(* IEC 61131-3 sources: std_i2980_v2.06_cp053/Source/IMM/ieccontrol/InjectionGeneral (part 15) *)

(* ---- ABMovePVCalib.pu ---- *)
(*
@h    ! WARNING !
@h    The Kemro K2 system (including software) only meets category B according to EN 954-1,
@h    thus it is not intended for usage in safety-relevant control applications in the field
@h    of personal safety (e.g. emergency stop).
@h    To implement potentially necessary safety-relevant control tasks, always use additional
@h    external safety devices that are intended for the particular purpose, and meet the necessary
@h    functional safety.
@h    For further information see EN 954-1 (EN ISO 13849-1) and/or the K2-x00 user manual, chapter
@h    "CE conformity, directives and standards".

In this AB the inject movements are realized.
This means inject movement with cutoff detection, inject movement in setup mode,
calibration for screw transducer (forward) and also the inject movement for auto purging

@FunctionID: S_KPIEC_PRINJ_01
@FunctionID: S_KPIEC_PRINJ_02
@FunctionID: S_KPIEC_CALTRANS_04

*)

IMPORT_OVER_LISTFILE
 GET_MY_FU_NAME
, SET_ALARM
, FCalculateCylinderSize
, FCalcScrewSize
, cLockGroupHeatingNozzle
, cLockGroupSafetyGateNozzle
, cLockGroupSafetyGateMold
, cLockGroupMotor
, nActive
, nInactive
, nSetup
, tnCalibState_Aborted
, tnCalibState_Error
, cValueChangeDuringCalibTooLow
, cMovePVCalib
, MAX_VOLTAGE
, cMoveBwd
, tnOperationMode
, tsVelPre
, tsMoveData
, KAPPL_LintabData3D
, KCTRL_Stable_Param
, tsCylinderData
, tsTraceLevel
, tsMoveCtrl
, ABPumpPressureVelocityCalib
, tsPumpCalibError
, tyCalibDevices
, tsDeviceId
, tyPumpData
, ABMovementRegister
, FBSetMovementState

END_IMPORT

ALGORITHM_BLOCK ABMovePVCalib #DUMMY_EDIT_BLOCK

SYSTEM_VAR
 sv_OperationMode : tnOperationMode;
 sv_rPressure : REAL;
 sv_rVelocity : REAL;
 sv_bOutputActive : BOOL (* Output is active *);
 sv_bPreOutputReady : BOOL (* PreOutput is ready *);
 sv_bTransducerError : BOOL;
 sv_bDoPumpPressureCalib : BOOL;
 sv_bDoPumpVelocityCalib : BOOL;
 sv_ConstPumpPressureVelocCalib : tsVelPre;
 sv_rScrewVelocity : REAL;
 sv_MovePVCalib : tsMoveData;
 sv_rActPressureHydr : REAL;
 sv_TmpLintab : KAPPL_LintabData3D;
 sv_rServoOutput : REAL;
 sv_ConstServoPressureVelocCalib : tsVelPre;
 sv_bPumpPreVelCalibAnotherStepN : BOOL;
 sv_bPumpPreVelCalibDone : BOOL;
 sv_rScrewPosition : REAL;
 sv_PressureStableParam : KCTRL_Stable_Param;
 sv_VelocityStableParam : KCTRL_Stable_Param;
 sv_CylinderData : tsCylinderData;
 sv_rScrewDiameter : REAL;
 sv_rTmpMaxAbsFlow : REAL;
 sv_TraceLevel : tsTraceLevel;
 sv_rScrewVolume : REAL;
 sv_rMaxVoltageVelocityPresCalib : REAL;
 sv_rMaxMeasurePositionRel : REAL;
 sv_PumpCalibError : tsPumpCalibError;
 sv_PumpCalibDevices : tyCalibDevices (* !!! device 1 - 20 reserved !!! *);
 sv_MoveDecompAftPlast : tsMoveData;
 sv_MoveInject : tsMoveData;
 sv_rScrewVelocityAbs : REAL (* screw velocity in mm/s *);
 sv_DeviceId : tsDeviceId;
 ai_Pressure : REAL;
 ai_SysPressure : REAL;
 sv_iCalibratingPump : DINT (* number of pump which is actually calibrating *);
 sv_PumpData : tyPumpData;
END_VAR

SYSTEM_OBJECT
 TaskInject : TASK;
 erSetupModeRequiredForCalib : ALARM;
END_OBJECT

VAR_EXTERNAL
 g_MoveCtrl : tsMoveCtrl;
END_VAR

VAR
 abPumpPressureVelocityCalib : ABPumpPressureVelocityCalib;
END_VAR

(*
This algorithm is necessary for registering the available movements
and the according parameters (Lockgroups, icon path, delay time, ....)
*)

ALGORITHM aRegister

VAR
 abInjectRegister : ABMovementRegister;
END_VAR
#BEGIN_EDIT_BLOCK
(**************************************** WARNING ********************************************
 *** The KEBA Kemro K2 System including software is not intended for safety control tasks! ***
 ***                       For further information see Comment tab!                        ***
 *********************************************************************************************)

//register inject movement
sv_MovePVCalib.LockGroups[1] := cLockGroupHeatingNozzle;
sv_MovePVCalib.LockGroups[2] := cLockGroupSafetyGateNozzle;
sv_MovePVCalib.LockGroups[3] := cLockGroupSafetyGateMold;
sv_MovePVCalib.LockGroups[4] := cLockGroupMotor;
sv_MovePVCalib.sIconPath := CONCAT(GET_MY_FU_NAME(),"\hmi\images\movScrewFwd.gif");

abInjectRegister.aRegister(@sv_MovePVCalib);

;#END_EDIT_BLOCK END_ALGORITHM

(*
This algorithm is responsible for executing the movement.
Depending on MoveId, OperationMode and activated transducer calibration the according
movement is executed.
The different actions contain the movement blocks and the according parameters.
*)

ALGORITHM aRun

VAR_INPUT
 bStop : BOOL (* flag if the movement should be stopped *);
END_VAR

VAR_OUTPUT
 bReady : BOOL (* information if movement is ready *);
END_VAR

VAR
 fbSetMovementState : FBSetMovementState;
 bError : BOOL;
 rSizeHydraulicCylinder : REAL;
 rSizeScrewCylinder : REAL;
 rTmpMaxAbsVel : REAL;
 iLastCalibratedPump : DINT;
END_VAR

(* IecGraph-Code *)

(* init step *)
INITIAL_STEP START:
AStart (P);
END_STEP

ACTION AStart: #BEGIN_EDIT_BLOCK
bReady := FALSE;
fbSetMovementState(MoveId   := g_MoveCtrl.pData^.MoveId,
                   MoveDir  := g_MoveCtrl.pData^.MoveDir,
                   State    := nActive);

;#END_EDIT_BLOCK END_ACTION (*AStart*)

(* steps *)
STEP S_InitMaxVoltage:
AInit (P);
END_STEP

STEP S_NotInSetupMode:
ANotInSetupMode (P);
END_STEP

ACTION ANotInSetupMode: #BEGIN_EDIT_BLOCK
SET_ALARM(erSetupModeRequiredForCalib);

;#END_EDIT_BLOCK END_ACTION (*ANotInSetupMode*)
STEP S_InjectPresVelCalib:
AResetCalibPressureVelocity (P);
APressureVelocityCalib (N);
ACalc (P0);
END_STEP

STEP S_Ready:
AReady (P);
END_STEP

ACTION AReady: #BEGIN_EDIT_BLOCK
bReady := TRUE;
fbSetMovementState(MoveId   := g_MoveCtrl.pData^.MoveId,
                   MoveDir  := g_MoveCtrl.pData^.MoveDir,
                   State    := nInactive);

;#END_EDIT_BLOCK END_ACTION (*AReady*)

(* transitions *)
GO_ON_TRANSITION TSetupMode (* TSetupMode *) FROM START TO S_InitMaxVoltage :=  #BEGIN_EDIT_BLOCK
sv_OperationMode = nSetup

;#END_EDIT_BLOCK
END_TRANSITION

TRANSITION Trans6 (* Trans6 *) FROM S_InitMaxVoltage TO S_InjectPresVelCalib :=  #BEGIN_EDIT_BLOCK
TRUE
;#END_EDIT_BLOCK
END_TRANSITION

GO_ON_TRANSITION TNotSetupMode (* TNotSetupMode *) FROM START TO S_NotInSetupMode :=  #BEGIN_EDIT_BLOCK
sv_OperationMode <> nSetup
;#END_EDIT_BLOCK
END_TRANSITION

GO_ON_TRANSITION Trans35 (* Trans35 *) FROM S_NotInSetupMode TO S_Ready :=  #BEGIN_EDIT_BLOCK
TRUE
;#END_EDIT_BLOCK
END_TRANSITION

TRANSITION TPVCalibDone (* TPVCalibDone *) FROM S_InjectPresVelCalib TO S_Ready :=  #BEGIN_EDIT_BLOCK
NOT abPumpPressureVelocityCalib.aRun.bActive
;#END_EDIT_BLOCK
END_TRANSITION

TRANSITION TReady (* TReady *) FROM S_Ready TO START :=  #BEGIN_EDIT_BLOCK
TRUE
;#END_EDIT_BLOCK
END_TRANSITION

(* end IecGraph-Code *)
(* sfc-code *)

(* stand alone actions *)
ACTION AResetCalibPressureVelocity: #BEGIN_EDIT_BLOCK
(**************************************** WARNING ********************************************
 *** The KEBA Kemro K2 System including software is not intended for safety control tasks! ***
 ***                       For further information see Comment tab!                        ***
 *********************************************************************************************)

bError := FALSE;
abPumpPressureVelocityCalib.aRun(bStart := FALSE);

;#END_EDIT_BLOCK END_ACTION (*AResetCalibPressureVelocity*)
ACTION ACalc: #BEGIN_EDIT_BLOCK
(**************************************** WARNING ********************************************
 *** The KEBA Kemro K2 System including software is not intended for safety control tasks! ***
 ***                       For further information see Comment tab!                        ***
 *********************************************************************************************)

IF sv_bPumpPreVelCalibDone AND NOT bError THEN
   rSizeHydraulicCylinder := FCalculateCylinderSize(CylinderData := sv_CylinderData, bSmallSize := sv_CylinderData.bUseSmallSize, bCalcHighPressSize := FALSE);
   rSizeScrewCylinder := FCalcScrewSize(rDiameter := sv_rScrewDiameter);

   // convert velocity from [cm^3/s] to [mm/s]
   rTmpMaxAbsVel := abPumpPressureVelocityCalib.aRun.rMaxVelocityAbs * 1000.0 / rSizeScrewCylinder;

   // convert velocity from [mm/s] to [l/min] in hydraulic volume
   sv_rTmpMaxAbsFlow := rTmpMaxAbsVel * rSizeHydraulicCylinder / 1000000.0 * 60.0;
END_IF;

;#END_EDIT_BLOCK END_ACTION (*ACalc*)
ACTION APressureVelocityCalib: #BEGIN_EDIT_BLOCK
(**************************************** WARNING ********************************************
 *** The KEBA Kemro K2 System including software is not intended for safety control tasks! ***
 ***                       For further information see Comment tab!                        ***
 *********************************************************************************************)

//output pressure in bar, velocity in % of Pump
abPumpPressureVelocityCalib.aRun(bStop := bStop OR sv_bTransducerError,
                                 bStart := TRUE,
                                 rActPosition := sv_rScrewPosition,
                                 rMaxPosition := sv_rScrewVolume,
                                 rActVel := sv_rScrewVelocity,
                                 rActPressure := sv_rActPressureHydr,
                                 bIsPressureCalib := sv_bDoPumpPressureCalib,
                                 bIsVelocityCalib := sv_bDoPumpVelocityCalib,
                                 bIsServoValveCalib := FALSE,
                                 bDirection := FALSE,
                                 dDelayTimePump := T#200ms,
                                 rLimitPositionFactor := sv_rMaxMeasurePositionRel,
                                 bActive => sv_bOutputActive,
                                 rOutputPre => sv_rPressure,
                                 rOutputVel => sv_rVelocity,
                                 rOutputServo => sv_rServoOutput,
                                 bPreOutputReached => sv_bPreOutputReady,
                                 bError => sv_PumpCalibError.bError,
                                 iErrorInfo => sv_PumpCalibError.iErrorInfo);

;#END_EDIT_BLOCK END_ACTION (*APressureVelocityCalib*)
ACTION AInit: #BEGIN_EDIT_BLOCK
(**************************************** WARNING ********************************************
 *** The KEBA Kemro K2 System including software is not intended for safety control tasks! ***
 ***                       For further information see Comment tab!                        ***
 *********************************************************************************************)

IF iLastCalibratedPump <> sv_iCalibratingPump THEN
   //get max voltages of the pump which should be calibrated
   abPumpPressureVelocityCalib.aInitMaxVoltages.rMaxVoltage := MAX_VOLTAGE;
   abPumpPressureVelocityCalib.aInitMaxVoltages.rMinVoltage := 0.0;
   abPumpPressureVelocityCalib.aInitMaxVoltages.prMaxVoltageVelocity := sv_PumpData[sv_iCalibratingPump].prMaxVoltageV;
   abPumpPressureVelocityCalib.aInitMaxVoltages.prMaxVoltagePressure := sv_PumpData[sv_iCalibratingPump].prMaxVoltageP;
   abPumpPressureVelocityCalib.aInitMaxVoltages.prMaxVoltageVelocityPresCalib := @sv_rMaxVoltageVelocityPresCalib;
   abPumpPressureVelocityCalib.aInitMaxVoltages();

   iLastCalibratedPump := sv_iCalibratingPump;
END_IF;

;#END_EDIT_BLOCK END_ACTION (*AInit*)
(* end sfc-code *)

END_ALGORITHM

ALGORITHM aInit

VAR_TEMP
 i : DINT;
END_VAR
#BEGIN_EDIT_BLOCK
(**************************************** WARNING ********************************************
 *** The KEBA Kemro K2 System including software is not intended for safety control tasks! ***
 ***                       For further information see Comment tab!                        ***
 *********************************************************************************************)

abPumpPressureVelocityCalib.aInit(pConst := @sv_ConstPumpPressureVelocCalib,
                                  pConstServo := @sv_ConstServoPressureVelocCalib,
                                  MoveId := cMovePVCalib,
                                  pTmpLintab := @sv_TmpLintab,
                                  pbPumpPreVelCalibAnotherStepN := @sv_bPumpPreVelCalibAnotherStepN,
                                  pbPumpPreVelCalibDone := @sv_bPumpPreVelCalibDone,
                                  pPressureStableParam := @sv_PressureStableParam,
                                  pVelocityStableParam := @sv_VelocityStableParam,
                                  debugInstanceName := 'PVCalib',
                                  debugTask := TaskInject,
                                  pbDebugCalibration := @sv_TraceLevel.bDebugCalibration);

//add calib information to sv_PumpCalibDevices - list
FOR i := 1 TO cMaxCalibDevices DO
   IF sv_PumpCalibDevices[i].DeviceId = sv_DeviceId THEN
      sv_PumpCalibDevices[i].pVelCalibStartPosMovement := @sv_MoveDecompAftPlast;
      sv_PumpCalibDevices[i].pVelCalibMovement := @sv_MovePVCalib;
      sv_PumpCalibDevices[i].pPresCalibStartPosMovement := @sv_MoveInject;
      sv_PumpCalibDevices[i].pPresCalibMovement := @sv_MovePVCalib;
      sv_PumpCalibDevices[i].prActVelocity := @sv_rScrewVelocityAbs;
      IF IS_LINKED(ai_Pressure) OR IS_LINKED(ai_SysPressure) THEN
         sv_PumpCalibDevices[i].prActPressure := @sv_rActPressureHydr;
      END_IF;
      EXIT;
   END_IF;
END_FOR;

;#END_EDIT_BLOCK END_ALGORITHM

END_ALGORITHM_BLOCK

#END_OF_IEC_PART

@Puma @IecEditor 6 120 @Pou 25
@@@BEG_Comment@@@
@h    ! WARNING !
@h    The Kemro K2 system (including software) only meets category B according to EN 954-1,
@h    thus it is not intended for usage in safety-relevant control applications in the field
@h    of personal safety (e.g. emergency stop).
@h    To implement potentially necessary safety-relevant control tasks, always use additional
@h    external safety devices that are intended for the particular purpose, and meet the necessary
@h    functional safety.
@h    For further information see EN 954-1 (EN ISO 13849-1) and/or the K2-x00 user manual, chapter
@h    "CE conformity, directives and standards".

In this AB the inject movements are realized.
This means inject movement with cutoff detection, inject movement in setup mode,
calibration for screw transducer (forward) and also the inject movement for auto purging

@FunctionID: S_KPIEC_PRINJ_01
@FunctionID: S_KPIEC_PRINJ_02
@FunctionID: S_KPIEC_CALTRANS_04

@@@END_Comment@@@

@BEG_Contents

@BEG_Func
@RT(17)FuncTreeContainer
4
@Var @RT(14)GET_MY_FU_NAME @RT(0) @T @T @DERIVED 0 @F @RT(22)KEBA_STANDARD_FUNCTION @F
@T
@BEG_Attrib
0 @RT(0) @RT(0)
@END_Attrib
1 1 @F @F @F @F

@Var @RT(9)SET_ALARM @RT(0) @T @T @DERIVED 0 @F @RT(23)KEBA_STANDARD_PROCEDURE @F
@T
@BEG_Attrib
0 @RT(0) @RT(0)
@END_Attrib
1 1 @F @F @F @F

@Var @RT(22)FCalculateCylinderSize @RT(0) @T @T @DERIVED 0 @F @RT(8)FUNCTION @F
@T
@BEG_Attrib
0 @RT(0) @RT(0)
@END_Attrib
1 1 @F @F @F @F

@Var @RT(14)FCalcScrewSize @RT(0) @T @T @DERIVED 0 @F @RT(8)FUNCTION @F
@T
@BEG_Attrib
0 @RT(0) @RT(0)
@END_Attrib
1 1 @F @F @F @F

@END_Func

@BEG_Const
@RT(18)ConstTreeContainer
13
@Var @RT(23)cLockGroupHeatingNozzle @RT(0) @T @F @DT @RT(4)DINT @RT(0) @T @T @BASIC 0 @F
@F @F
@T
@BEG_Attrib
0 @RT(2)63 @RT(35)Members: Injection, Plast, Suckback
@END_Attrib
1 1 @F @F @F @F

@Var @RT(26)cLockGroupSafetyGateNozzle @RT(0) @T @F @DT @RT(4)DINT @RT(0) @T @T @BASIC 0 @F
@F @F
@T
@BEG_Attrib
0 @RT(2)62 @RT(59)Members: Nozzle Forward, Injection, Plast, Intrusion, Purge
@END_Attrib
1 1 @F @F @F @F

@Var @RT(24)cLockGroupSafetyGateMold @RT(0) @T @F @DT @RT(4)DINT @RT(0) @T @T @BASIC 0 @F
@F @F
@T
@BEG_Attrib
0 @RT(2)61 @RT(73)Members: Mold Close, Mold Hight Forward, Auto Mold Hight, Core In, Inject
@END_Attrib
1 1 @F @F @F @F

@Var @RT(15)cLockGroupMotor @RT(0) @T @F @DT @RT(4)DINT @RT(0) @T @T @BASIC 0 @F
@F @F
@T
@BEG_Attrib
0 @RT(2)69 @RT(56)Members: Mold, Ejector, Cores, Injection, Plast, Purge,
@END_Attrib
1 1 @F @F @F @F

@Var @RT(7)nActive @RT(0) @T @T @DERIVED 0 @F @RT(16)tnActiveInactive @F
@T
@BEG_Attrib
0 @RT(1)1 @RT(0)
@END_Attrib
1 1 @F @F @F @F

@Var @RT(9)nInactive @RT(0) @T @T @DERIVED 0 @F @RT(16)tnActiveInactive @F
@T
@BEG_Attrib
0 @RT(1)0 @RT(0)
@END_Attrib
1 1 @F @F @F @F

@Var @RT(6)nSetup @RT(0) @T @T @DERIVED 0 @F @RT(15)tnOperationMode @F
@T
@BEG_Attrib
0 @RT(1)0 @RT(36)Setup mode only for service engineer
@END_Attrib
1 1 @F @F @F @F

@Var @RT(20)tnCalibState_Aborted @RT(0) @T @T @DERIVED 0 @F @RT(12)tnCalibState @F
@T
@BEG_Attrib
0 @RT(1)4 @RT(19)calibration aborted
@END_Attrib
1 1 @F @F @F @F

@Var @RT(18)tnCalibState_Error @RT(0) @T @T @DERIVED 0 @F @RT(12)tnCalibState @F
@T
@BEG_Attrib
0 @RT(1)3 @RT(32)error occured during calibration
@END_Attrib
1 1 @F @F @F @F

@Var @RT(29)cValueChangeDuringCalibTooLow @RT(0) @T @F @DT @RT(4)DINT @RT(0) @T @T @BASIC 0 @F
@F @F
@T
@BEG_Attrib
0 @RT(4)-510 @RT(94)no or too low value change (velocity, pressure, rpm, ..) detected during calibration procedure
@END_Attrib
1 1 @F @F @F @F

@Var @RT(12)cMovePVCalib @RT(0) @T @F @DT @RT(4)DINT @RT(0) @T @T @BASIC 0 @F
@F @F
@T
@BEG_Attrib
0 @RT(2)38 @RT(38)injection movement with voltage output
@END_Attrib
1 1 @F @F @F @F

@Var @RT(11)MAX_VOLTAGE @RT(0) @T @F @DT @RT(4)REAL @RT(0) @T @T @BASIC 0 @F
@F @F
@T
@BEG_Attrib
0 @RT(4)10.0 @RT(0)
@END_Attrib
1 1 @F @F @F @F

@Var @RT(8)cMoveBwd @RT(0) @T @F @DT @RT(4)DINT @RT(0) @T @T @BASIC 0 @F
@F @F
@T
@BEG_Attrib
0 @RT(2)11 @RT(17)movement backward
@END_Attrib
1 1 @F @F @F @F

@END_Const

@BEG_Export

@BEG_Kind
@ALGORITHM_BLOCK @RT(13)ABMovePVCalib @STRUCTURED_TEXT
@RT(0) @RT(0) @RT(0)
@END_Kind

@BEG_Dcl
@RT(16)DclTreeContainer
41
@Var @RT(16)sv_OperationMode @RT(0) @T @T @DERIVED 0 @T @T @DT @RT(15)tnOperationMode @RT(0) @T @T @UNKNOWN 0 @F
@F @F
@T
@BEG_Attrib
3 @RT(0) @RT(0) @RT(0)
@END_Attrib
1 8 @F @F @F @F

@Var @RT(12)sv_rPressure @RT(0) @T @F @DT @RT(4)REAL @RT(0) @T @T @BASIC 0 @F
@F @F
@T
@BEG_Attrib
3 @RT(0) @RT(0) @RT(0)
@END_Attrib
1 8 @F @F @F @F

@Var @RT(12)sv_rVelocity @RT(0) @T @F @DT @RT(4)REAL @RT(0) @T @T @BASIC 0 @F
@F @F
@T
@BEG_Attrib
3 @RT(0) @RT(0) @RT(0)
@END_Attrib
1 8 @F @F @F @F

@Var @RT(16)sv_bOutputActive @RT(0) @T @F @DT @RT(4)BOOL @RT(0) @T @T @BASIC 0 @F
@F @F
@T
@BEG_Attrib
3 @RT(0) @RT(16)Output is active @RT(0)
@END_Attrib
1 8 @F @F @F @F

@Var @RT(18)sv_bPreOutputReady @RT(0) @T @F @DT @RT(4)BOOL @RT(0) @T @T @BASIC 0 @F
@F @F
@T
@BEG_Attrib
3 @RT(0) @RT(18)PreOutput is ready @RT(0)
@END_Attrib
1 8 @F @F @F @F

@Var @RT(19)sv_bTransducerError @RT(0) @T @F @DT @RT(4)BOOL @RT(0) @T @T @BASIC 0 @F
@F @F
@T
@BEG_Attrib
3 @RT(0) @RT(0) @RT(0)
@END_Attrib
1 8 @F @F @F @F

@Var @RT(23)sv_bDoPumpPressureCalib @RT(0) @T @F @DT @RT(4)BOOL @RT(0) @T @T @BASIC 0 @F
@F @F
@T
@BEG_Attrib
3 @RT(0) @RT(0) @RT(0)
@END_Attrib
1 8 @F @F @F @F

@Var @RT(23)sv_bDoPumpVelocityCalib @RT(0) @T @F @DT @RT(4)BOOL @RT(0) @T @T @BASIC 0 @F
@F @F
@T
@BEG_Attrib
3 @RT(0) @RT(0) @RT(0)
@END_Attrib
1 8 @F @F @F @F

@Var @RT(30)sv_ConstPumpPressureVelocCalib @RT(0) @T @T @DERIVED 0 @T @T @DT @RT(8)tsVelPre @RT(0) @T @T @UNKNOWN 0 @F
@F @F
@T
@BEG_Attrib
3 @RT(0) @RT(0) @RT(0)
@END_Attrib
1 8 @F @F @F @F

@Var @RT(17)sv_rScrewVelocity @RT(0) @T @F @DT @RT(4)REAL @RT(0) @T @T @BASIC 0 @F
@F @F
@T
@BEG_Attrib
3 @RT(0) @RT(0) @RT(0)
@END_Attrib
1 8 @F @F @F @F

@Var @RT(14)sv_MovePVCalib @RT(0) @T @T @DERIVED 0 @T @T @DT @RT(10)tsMoveData @RT(0) @T @T @UNKNOWN 0 @F
@F @F
@T
@BEG_Attrib
3 @RT(0) @RT(0) @RT(0)
@END_Attrib
1 8 @F @F @F @F

@Var @RT(19)sv_rActPressureHydr @RT(0) @T @F @DT @RT(4)REAL @RT(0) @T @T @BASIC 0 @F
@F @F
@T
@BEG_Attrib
3 @RT(0) @RT(0) @RT(0)
@END_Attrib
1 8 @F @F @F @F

@Var @RT(12)sv_TmpLintab @RT(0) @T @T @DERIVED 0 @T @T @DT @RT(18)KAPPL_LintabData3D @RT(0) @T @T @UNKNOWN 0 @F
@F @F
@T
@BEG_Attrib
3 @RT(0) @RT(0) @RT(0)
@END_Attrib
1 8 @F @F @F @F

@Var @RT(15)sv_rServoOutput @RT(0) @T @F @DT @RT(4)REAL @RT(0) @T @T @BASIC 0 @F
@F @F
@T
@BEG_Attrib
3 @RT(0) @RT(0) @RT(0)
@END_Attrib
1 8 @F @F @F @F

@Var @RT(31)sv_ConstServoPressureVelocCalib @RT(0) @T @T @DERIVED 0 @T @T @DT @RT(8)tsVelPre @RT(0) @T @T @UNKNOWN 0 @F
@F @F
@T
@BEG_Attrib
3 @RT(0) @RT(0) @RT(0)
@END_Attrib
1 8 @F @F @F @F

@Var @RT(31)sv_bPumpPreVelCalibAnotherStepN @RT(0) @T @F @DT @RT(4)BOOL @RT(0) @T @T @BASIC 0 @F
@F @F
@T
@BEG_Attrib
3 @RT(0) @RT(0) @RT(0)
@END_Attrib
1 8 @F @F @F @F

@Var @RT(23)sv_bPumpPreVelCalibDone @RT(0) @T @F @DT @RT(4)BOOL @RT(0) @T @T @BASIC 0 @F
@F @F
@T
@BEG_Attrib
3 @RT(0) @RT(0) @RT(0)
@END_Attrib
1 8 @F @F @F @F

@Var @RT(17)sv_rScrewPosition @RT(0) @T @F @DT @RT(4)REAL @RT(0) @T @T @BASIC 0 @F
@F @F
@T
@BEG_Attrib
3 @RT(0) @RT(0) @RT(0)
@END_Attrib
1 8 @F @F @F @F

@Var @RT(22)sv_PressureStableParam @RT(0) @T @T @DERIVED 0 @T @T @DT @RT(18)KCTRL_Stable_Param @RT(0) @T @T @UNKNOWN 0 @F
@F @F
@T
@BEG_Attrib
3 @RT(0) @RT(0) @RT(0)
@END_Attrib
1 8 @F @F @F @F

@Var @RT(22)sv_VelocityStableParam @RT(0) @T @T @DERIVED 0 @T @T @DT @RT(18)KCTRL_Stable_Param @RT(0) @T @T @UNKNOWN 0 @F
@F @F
@T
@BEG_Attrib
3 @RT(0) @RT(0) @RT(0)
@END_Attrib
1 8 @F @F @F @F

@Var @RT(15)sv_CylinderData @RT(0) @T @T @DERIVED 0 @T @T @DT @RT(14)tsCylinderData @RT(0) @T @T @UNKNOWN 0 @F
@F @F
@T
@BEG_Attrib
3 @RT(0) @RT(0) @RT(0)
@END_Attrib
1 8 @F @F @F @F

@Var @RT(17)sv_rScrewDiameter @RT(0) @T @F @DT @RT(4)REAL @RT(0) @T @T @BASIC 0 @F
@F @F
@T
@BEG_Attrib
3 @RT(0) @RT(0) @RT(0)
@END_Attrib
1 8 @F @F @F @F

@Var @RT(17)sv_rTmpMaxAbsFlow @RT(0) @T @F @DT @RT(4)REAL @RT(0) @T @T @BASIC 0 @F
@F @F
@T
@BEG_Attrib
3 @RT(0) @RT(0) @RT(0)
@END_Attrib
1 8 @F @F @F @F

@Var @RT(13)sv_TraceLevel @RT(0) @T @T @DERIVED 0 @T @T @DT @RT(12)tsTraceLevel @RT(0) @T @T @UNKNOWN 0 @F
@F @F
@T
@BEG_Attrib
3 @RT(0) @RT(0) @RT(0)
@END_Attrib
1 8 @F @F @F @F

@Var @RT(15)sv_rScrewVolume @RT(0) @T @F @DT @RT(4)REAL @RT(0) @T @T @BASIC 0 @F
@F @F
@T
@BEG_Attrib
3 @RT(0) @RT(0) @RT(0)
@END_Attrib
1 8 @F @F @F @F

@Var @RT(31)sv_rMaxVoltageVelocityPresCalib @RT(0) @T @F @DT @RT(4)REAL @RT(0) @T @T @BASIC 0 @F
@F @F
@T
@BEG_Attrib
3 @RT(0) @RT(0) @RT(0)
@END_Attrib
1 8 @F @F @F @F

@Var @RT(25)sv_rMaxMeasurePositionRel @RT(0) @T @F @DT @RT(4)REAL @RT(0) @T @T @BASIC 0 @F
@F @F
@T
@BEG_Attrib
3 @RT(0) @RT(0) @RT(0)
@END_Attrib
1 8 @F @F @F @F

@Var @RT(10)TaskInject @RT(0) @T @F @DT @RT(4)TASK @RT(0) @T @T @BASIC 0 @F
@F @F
@T
@BEG_Attrib
3 @RT(0) @RT(0) @RT(0)
@END_Attrib
1 7 @F @F @F @F

@Var @RT(27)erSetupModeRequiredForCalib @RT(0) @T @F @DT @RT(5)ALARM @RT(0) @T @T @BASIC 0 @F
@F @F
@T
@BEG_Attrib
3 @RT(0) @RT(0) @RT(0)
@END_Attrib
1 7 @F @F @F @F

@Var @RT(10)g_MoveCtrl @RT(0) @T @T @DERIVED 0 @T @T @DT @RT(10)tsMoveCtrl @RT(0) @T @T @UNKNOWN 0 @F
@F @F
@T
@BEG_Attrib
3 @RT(0) @RT(0) @RT(0)
@END_Attrib
1 6 @F @F @F @F

@Var @RT(27)abPumpPressureVelocityCalib @RT(0) @T @T @DERIVED 0 @T @T @DT @RT(27)ABPumpPressureVelocityCalib @RT(0) @T @T @UNKNOWN 0 @F
@F @F
@T
@BEG_Attrib
3 @RT(0) @RT(0) @RT(0)
@END_Attrib
1 0 @F @F @F @F

@Var @RT(17)sv_PumpCalibError @RT(0) @T @T @DERIVED 0 @T @T @DT @RT(16)tsPumpCalibError @RT(0) @T @T @UNKNOWN 0 @F
@F @F
@T
@BEG_Attrib
3 @RT(0) @RT(0) @RT(0)
@END_Attrib
1 8 @F @F @F @F

@Var @RT(19)sv_PumpCalibDevices @RT(0) @T @T @DERIVED 0 @T @T @DT @RT(14)tyCalibDevices @RT(0) @T @T @UNKNOWN 0 @F
@F @F
@T
@BEG_Attrib
3 @RT(0) @RT(30)!!! device 1 - 20 reserved !!! @RT(0)
@END_Attrib
1 8 @F @F @F @F

@Var @RT(21)sv_MoveDecompAftPlast @RT(0) @T @T @DERIVED 0 @T @T @DT @RT(10)tsMoveData @RT(0) @T @T @UNKNOWN 0 @F
@F @F
@T
@BEG_Attrib
3 @RT(0) @RT(0) @RT(0)
@END_Attrib
1 8 @F @F @F @F

@Var @RT(13)sv_MoveInject @RT(0) @T @T @DERIVED 0 @T @T @DT @RT(10)tsMoveData @RT(0) @T @T @UNKNOWN 0 @F
@F @F
@T
@BEG_Attrib
3 @RT(0) @RT(0) @RT(0)
@END_Attrib
1 8 @F @F @F @F

@Var @RT(20)sv_rScrewVelocityAbs @RT(0) @T @F @DT @RT(4)REAL @RT(0) @T @T @BASIC 0 @F
@F @F
@T
@BEG_Attrib
3 @RT(0) @RT(22)screw velocity in mm/s @RT(0)
@END_Attrib
1 8 @F @F @F @F

@Var @RT(11)sv_DeviceId @RT(0) @T @T @DERIVED 0 @T @T @DT @RT(10)tsDeviceId @RT(0) @T @T @UNKNOWN 0 @F
@F @F
@T
@BEG_Attrib
3 @RT(0) @RT(0) @RT(0)
@END_Attrib
1 8 @F @F @F @F

@Var @RT(11)ai_Pressure @RT(0) @T @F @DT @RT(4)REAL @RT(0) @T @T @BASIC 0 @F
@F @F
@T
@BEG_Attrib
3 @RT(0) @RT(0) @RT(0)
@END_Attrib
1 8 @F @F @F @F

@Var @RT(14)ai_SysPressure @RT(0) @T @F @DT @RT(4)REAL @RT(0) @T @T @BASIC 0 @F
@F @F
@T
@BEG_Attrib
3 @RT(0) @RT(0) @RT(0)
@END_Attrib
1 8 @F @F @F @F

@Var @RT(19)sv_iCalibratingPump @RT(0) @T @F @DT @RT(4)DINT @RT(0) @T @T @BASIC 0 @F
@F @F
@T
@BEG_Attrib
3 @RT(0) @RT(44)number of pump which is actually calibrating @RT(0)
@END_Attrib
1 8 @F @F @F @F

@Var @RT(11)sv_PumpData @RT(0) @T @T @DERIVED 0 @F @RT(10)tyPumpData @F
@T
@BEG_Attrib
3 @RT(0) @RT(0) @RT(0)
@END_Attrib
1 8 @F @F @F @F

@END_Dcl

@END_Export

@BEG_Body

3

@BEG_Export

@BEG_Algo
@ALGORITHM @RT(9)aRegister @STRUCTURED_TEXT
@RT(0) @RT(0) @RT(0) @F @F
@END_Algo

@BEG_Dcl
@RT(16)DclTreeContainer
1
@Var @RT(16)abInjectRegister @RT(0) @T @T @DERIVED 0 @T @T @DT @RT(18)ABMovementRegister @RT(0) @T @T @UNKNOWN 0 @F
@F @F
@T
@BEG_Attrib
3 @RT(0) @RT(0) @RT(0)
@END_Attrib
1 0 @F @F @F @F

@END_Dcl

@END_Export

@BEG_Export

@BEG_Algo
@ALGORITHM @RT(4)aRun @SEQUENTIAL_FLOW_CHART
@RT(0) @RT(0) @RT(0) @F @F
@END_Algo

@BEG_Dcl
@RT(16)DclTreeContainer
8
@Var @RT(5)bStop @RT(0) @T @F @DT @RT(4)BOOL @RT(0) @T @T @BASIC 0 @F
@F @F
@T
@BEG_Attrib
3 @RT(0) @RT(38)flag if the movement should be stopped @RT(0)
@END_Attrib
1 1 @F @F @F @F

@Var @RT(6)bReady @RT(0) @T @F @DT @RT(4)BOOL @RT(0) @T @T @BASIC 0 @F
@F @F
@T
@BEG_Attrib
3 @RT(0) @RT(32)information if movement is ready @RT(0)
@END_Attrib
1 3 @F @F @F @F

@Var @RT(18)fbSetMovementState @RT(0) @T @T @DERIVED 0 @T @T @DT @RT(18)FBSetMovementState @RT(0) @T @T @UNKNOWN 0 @F
@F @F
@T
@BEG_Attrib
3 @RT(0) @RT(0) @RT(0)
@END_Attrib
1 0 @F @F @F @F

@Var @RT(6)bError @RT(0) @T @F @DT @RT(4)BOOL @RT(0) @T @T @BASIC 0 @F
@F @F
@T
@BEG_Attrib
3 @RT(0) @RT(0) @RT(0)
@END_Attrib
1 0 @F @F @F @F

@Var @RT(22)rSizeHydraulicCylinder @RT(0) @T @F @DT @RT(4)REAL @RT(0) @T @T @BASIC 0 @F
@F @F
@T
@BEG_Attrib
3 @RT(0) @RT(0) @RT(0)
@END_Attrib
1 0 @F @F @F @F

@Var @RT(18)rSizeScrewCylinder @RT(0) @T @F @DT @RT(4)REAL @RT(0) @T @T @BASIC 0 @F
@F @F
@T
@BEG_Attrib
3 @RT(0) @RT(0) @RT(0)
@END_Attrib
1 0 @F @F @F @F

@Var @RT(13)rTmpMaxAbsVel @RT(0) @T @F @DT @RT(4)REAL @RT(0) @T @T @BASIC 0 @F
@F @F
@T
@BEG_Attrib
3 @RT(0) @RT(0) @RT(0)
@END_Attrib
1 0 @F @F @F @F

@Var @RT(19)iLastCalibratedPump @RT(0) @T @F @DT @RT(4)DINT @RT(0) @T @T @BASIC 0 @F
@F @F
@T
@BEG_Attrib
3 @RT(0) @RT(0) @RT(0)
@END_Attrib
1 0 @F @F @F @F

@END_Dcl

@END_Export

@BEG_Export

@BEG_Algo
@ALGORITHM @RT(5)aInit @STRUCTURED_TEXT
@RT(0) @RT(0) @RT(0) @F @F
@END_Algo

@BEG_Dcl
@RT(16)DclTreeContainer
1
@Var @RT(1)i @RT(0) @T @F @DT @RT(4)DINT @RT(0) @T @T @BASIC 0 @F
@F @F
@T
@BEG_Attrib
3 @RT(0) @RT(0) @RT(0)
@END_Attrib
1 4 @F @F @F @F

@END_Dcl

@END_Export

@BEG_Body
@TL(15)
(**************************************** WARNING ********************************************
 *** The KEBA Kemro K2 System including software is not intended for safety control tasks! ***
 ***                       For further information see Comment tab!                        ***
 *********************************************************************************************)

//register inject movement
sv_MovePVCalib.LockGroups[1] := cLockGroupHeatingNozzle;
sv_MovePVCalib.LockGroups[2] := cLockGroupSafetyGateNozzle;
sv_MovePVCalib.LockGroups[3] := cLockGroupSafetyGateMold;
sv_MovePVCalib.LockGroups[4] := cLockGroupMotor;
sv_MovePVCalib.sIconPath := CONCAT(GET_MY_FU_NAME(),"\hmi\images\movScrewFwd.gif");

abInjectRegister.aRegister(@sv_MovePVCalib);

@END_Body

@@@BEG_Comment@@@
@TL(2)
This algorithm is necessary for registering the available movements
and the according parameters (Lockgroups, icon path, delay time, ....)
@@@END_Comment@@@

@BEG_SfcBody
8 6 6

@BEG_SfcData 2
@StepSeq @RT(4)sseq @F 1
@Loop @RT(4)loop @F 2
@StepSeq @RT(4)sseq @F 5
@Step @RT(5)START @F @T @F @F @RT(0) @F
@AcbCont @RT(7)unnamed @F 1
@Acb @RT(6)AStart @F @T @RT(1)P @RT(0) @F @F @T @TL(5)
bReady := FALSE;
fbSetMovementState(MoveId   := g_MoveCtrl.pData^.MoveId,
                   MoveDir  := g_MoveCtrl.pData^.MoveDir,
                   State    := nActive);

@F

@AltBranch @RT(3)alt @F 2
@TransSeq @RT(4)tseq @F 3
@Trans @RT(10)TSetupMode @F @T @F @F @T @F @TL(3)
sv_OperationMode = nSetup

@RT(10)TSetupMode @F
@Step @RT(16)S_InitMaxVoltage @F @F @F @F @RT(0) @F
@AcbCont @RT(7)unnamed @F 1
@Acb @RT(5)AInit @F @F @RT(1)P @RT(0) @F @F @F @F

@Trans @RT(6)Trans6 @F @T @F @F @T @T @TL(2)
TRUE

@RT(6)Trans6 @F

@TransSeq @RT(4)tseq @F 4
@Trans @RT(13)TNotSetupMode @F @T @F @F @T @F @TL(2)
sv_OperationMode <> nSetup

@RT(13)TNotSetupMode @F
@Step @RT(16)S_NotInSetupMode @F @F @F @F @RT(0) @F
@AcbCont @RT(7)unnamed @F 1
@Acb @RT(15)ANotInSetupMode @F @T @RT(1)P @RT(0) @F @F @T @TL(2)
SET_ALARM(erSetupModeRequiredForCalib);

@F

@Trans @RT(7)Trans35 @F @T @F @F @T @F @TL(2)
TRUE

@RT(7)Trans35 @F
@Goto @RT(7)S_Ready @F @F

@Step @RT(20)S_InjectPresVelCalib @F @F @F @F @RT(0) @F
@AcbCont @RT(7)unnamed @F 3
@Acb @RT(27)AResetCalibPressureVelocity @F @F @RT(1)P @RT(0) @F @F @F @F
@Acb @RT(22)APressureVelocityCalib @F @F @RT(1)N @RT(0) @F @F @F @F
@Acb @RT(5)ACalc @F @F @RT(2)P0 @RT(0) @F @F @F @F

@Trans @RT(12)TPVCalibDone @F @T @F @F @T @T @TL(2)
NOT abPumpPressureVelocityCalib.aRun.bActive

@RT(12)TPVCalibDone @F
@Step @RT(7)S_Ready @F @F @T @F @RT(0) @F
@AcbCont @RT(7)unnamed @F 1
@Acb @RT(6)AReady @F @T @RT(1)P @RT(0) @F @F @T @TL(5)
bReady := TRUE;
fbSetMovementState(MoveId   := g_MoveCtrl.pData^.MoveId,
                   MoveDir  := g_MoveCtrl.pData^.MoveDir,
                   State    := nInactive);

@F

@Trans @RT(6)TReady @F @T @T @T @T @T @TL(2)
TRUE

@RT(6)TReady @F

@END_SfcData
@SaActions 4
@SaText @RT(27)AResetCalibPressureVelocity 1 @TL(8)
(**************************************** WARNING ********************************************
 *** The KEBA Kemro K2 System including software is not intended for safety control tasks! ***
 ***                       For further information see Comment tab!                        ***
 *********************************************************************************************)

bError := FALSE;
abPumpPressureVelocityCalib.aRun(bStart := FALSE);

@SaText @RT(5)ACalc 1 @TL(17)
(**************************************** WARNING ********************************************
 *** The KEBA Kemro K2 System including software is not intended for safety control tasks! ***
 ***                       For further information see Comment tab!                        ***
 *********************************************************************************************)

IF sv_bPumpPreVelCalibDone AND NOT bError THEN
   rSizeHydraulicCylinder := FCalculateCylinderSize(CylinderData := sv_CylinderData, bSmallSize := sv_CylinderData.bUseSmallSize, bCalcHighPressSize := FALSE);
   rSizeScrewCylinder := FCalcScrewSize(rDiameter := sv_rScrewDiameter);

   // convert velocity from [cm^3/s] to [mm/s]
   rTmpMaxAbsVel := abPumpPressureVelocityCalib.aRun.rMaxVelocityAbs * 1000.0 / rSizeScrewCylinder;

   // convert velocity from [mm/s] to [l/min] in hydraulic volume
   sv_rTmpMaxAbsFlow := rTmpMaxAbsVel * rSizeHydraulicCylinder / 1000000.0 * 60.0;
END_IF;

@SaText @RT(22)APressureVelocityCalib 1 @TL(26)
(**************************************** WARNING ********************************************
 *** The KEBA Kemro K2 System including software is not intended for safety control tasks! ***
 ***                       For further information see Comment tab!                        ***
 *********************************************************************************************)

//output pressure in bar, velocity in % of Pump
abPumpPressureVelocityCalib.aRun(bStop := bStop OR sv_bTransducerError,
                                 bStart := TRUE,
                                 rActPosition := sv_rScrewPosition,
                                 rMaxPosition := sv_rScrewVolume,
                                 rActVel := sv_rScrewVelocity,
                                 rActPressure := sv_rActPressureHydr,
                                 bIsPressureCalib := sv_bDoPumpPressureCalib,
                                 bIsVelocityCalib := sv_bDoPumpVelocityCalib,
                                 bIsServoValveCalib := FALSE,
                                 bDirection := FALSE,
                                 dDelayTimePump := T#200ms,
                                 rLimitPositionFactor := sv_rMaxMeasurePositionRel,
                                 bActive => sv_bOutputActive,
                                 rOutputPre => sv_rPressure,
                                 rOutputVel => sv_rVelocity,
                                 rOutputServo => sv_rServoOutput,
                                 bPreOutputReached => sv_bPreOutputReady,
                                 bError => sv_PumpCalibError.bError,
                                 iErrorInfo => sv_PumpCalibError.iErrorInfo);

@SaText @RT(5)AInit 1 @TL(20)
(**************************************** WARNING ********************************************
 *** The KEBA Kemro K2 System including software is not intended for safety control tasks! ***
 ***                       For further information see Comment tab!                        ***
 *********************************************************************************************)

IF iLastCalibratedPump <> sv_iCalibratingPump THEN
   //get max voltages of the pump which should be calibrated
   abPumpPressureVelocityCalib.aInitMaxVoltages.rMaxVoltage := MAX_VOLTAGE;
   abPumpPressureVelocityCalib.aInitMaxVoltages.rMinVoltage := 0.0;
   abPumpPressureVelocityCalib.aInitMaxVoltages.prMaxVoltageVelocity := sv_PumpData[sv_iCalibratingPump].prMaxVoltageV;
   abPumpPressureVelocityCalib.aInitMaxVoltages.prMaxVoltagePressure := sv_PumpData[sv_iCalibratingPump].prMaxVoltageP;
   abPumpPressureVelocityCalib.aInitMaxVoltages.prMaxVoltageVelocityPresCalib := @sv_rMaxVoltageVelocityPresCalib;
   abPumpPressureVelocityCalib.aInitMaxVoltages();

   iLastCalibratedPump := sv_iCalibratingPump;
END_IF;

@SaTrans 0
@SaExits 0
@END_SfcBody

@@@BEG_Comment@@@
@TL(4)
This algorithm is responsible for executing the movement.
Depending on MoveId, OperationMode and activated transducer calibration the according
movement is executed.
The different actions contain the movement blocks and the according parameters.
@@@END_Comment@@@

@BEG_Body
@TL(37)
(**************************************** WARNING ********************************************
 *** The KEBA Kemro K2 System including software is not intended for safety control tasks! ***
 ***                       For further information see Comment tab!                        ***
 *********************************************************************************************)

abPumpPressureVelocityCalib.aInit(pConst := @sv_ConstPumpPressureVelocCalib,
                                  pConstServo := @sv_ConstServoPressureVelocCalib,
                                  MoveId := cMovePVCalib,
                                  pTmpLintab := @sv_TmpLintab,
                                  pbPumpPreVelCalibAnotherStepN := @sv_bPumpPreVelCalibAnotherStepN,
                                  pbPumpPreVelCalibDone := @sv_bPumpPreVelCalibDone,
                                  pPressureStableParam := @sv_PressureStableParam,
                                  pVelocityStableParam := @sv_VelocityStableParam,
                                  debugInstanceName := 'PVCalib',
                                  debugTask := TaskInject,
                                  pbDebugCalibration := @sv_TraceLevel.bDebugCalibration);

//add calib information to sv_PumpCalibDevices - list
FOR i := 1 TO cMaxCalibDevices DO
   IF sv_PumpCalibDevices[i].DeviceId = sv_DeviceId THEN
      sv_PumpCalibDevices[i].pVelCalibStartPosMovement := @sv_MoveDecompAftPlast;
      sv_PumpCalibDevices[i].pVelCalibMovement := @sv_MovePVCalib;
      sv_PumpCalibDevices[i].pPresCalibStartPosMovement := @sv_MoveInject;
      sv_PumpCalibDevices[i].pPresCalibMovement := @sv_MovePVCalib;
      sv_PumpCalibDevices[i].prActVelocity := @sv_rScrewVelocityAbs;
      IF IS_LINKED(ai_Pressure) OR IS_LINKED(ai_SysPressure) THEN
         sv_PumpCalibDevices[i].prActPressure := @sv_rActPressureHydr;
      END_IF;
      EXIT;
   END_IF;
END_FOR;

@END_Body

@@@BEG_Comment@@@
@TL(0)

@@@END_Comment@@@
@END_Body

@END_Contents

(* ---- ABODCFunctions.pu ---- *)
(*
@h    ! WARNING !
@h    The Kemro K2 system (including software) only meets category B according to EN 954-1,
@h    thus it is not intended for usage in safety-relevant control applications in the field
@h    of personal safety (e.g. emergency stop).
@h    To implement potentially necessary safety-relevant control tasks, always use additional
@h    external safety devices that are intended for the particular purpose, and meet the necessary
@h    functional safety.
@h    For further information see EN 954-1 (EN ISO 13849-1) and/or the K2-x00 user manual, chapter
@h    "CE conformity, directives and standards".

Following functions are implemented in this AB
- registration of dummy movments for begin/end inject/plast sequence
- trigger new creation of machine sequence
- set/reset activated flags for intrusion and cold drop

@FunctionID: S_FU_05
@FunctionID: S_FU_04
@FunctionID: S_ALLG_09
*)

IMPORT_OVER_LISTFILE
 cMaxIntermediateConditions
, tsMoveData
, tsIntrusionParam
, tsColdDropParams
, tyInstanceListArrayDecomp
, ABMovementRegister
, FBUpdateEditorProperties

END_IMPORT

ALGORITHM_BLOCK ABODCFunctions #DUMMY_EDIT_BLOCK

SYSTEM_VAR
 sv_bInitStart : BOOL;
 sv_MoveBeginInjectSequence : tsMoveData;
 sv_MoveEndInjectSequence : tsMoveData;
 sv_MoveBeginPlastSequence : tsMoveData;
 sv_MoveEndPlastSequence : tsMoveData;
 sv_IntrusionSettings : tsIntrusionParam;
 sv_bProgramSwitchChanged : BOOL (* TRUE if ODC sequence should be reinitialized because a program switch changed *);
 sv_ColdDropSettings : tsColdDropParams;
 sv_dDurationInjectAndHold : TIME (* Duration of inject + hold *);
 sv_bHoldActive : BOOL (* TRUE: holding is active; attention: SV is resetted after end of inject movement *);
 sv_bInjectActive : BOOL (* Injection is active *);
 sv_InstanceDataDecompInterPos : tyInstanceListArrayDecomp;
 sv_bInitDone : BOOL;
 sv_MoveIntrusion : tsMoveData;
 sv_bUseProgramSwitches : BOOL (* TRUE: create sequence by using program switches; FALSE: use sequence from ODC editor *);
 sv_MoveColdDrop : tsMoveData;
END_VAR

SYSTEM_OBJECT
 PU_Task_7 : TASK;
 PU_Task_13 : TASK;
 TaskSlow : TASK;
END_OBJECT

(*
registers the following dummy - movements:
- begin of inject sequence
- end of inject sequence
- begin of plast sequence
- end of plast sequence
*)

POSTUPDATE_ALGORITHM pInitStart ON PU_Task_7 WITH sv_bInitStart

VAR
 abBeginInjSequenceRegister : ABMovementRegister;
 abEndInjSequenceRegister : ABMovementRegister;
 abBeginPlastSequenceRegister : ABMovementRegister;
 abEndPlastSequenceRegister : ABMovementRegister;
END_VAR
#BEGIN_EDIT_BLOCK
(**************************************** WARNING ********************************************
 *** The KEBA Kemro K2 System including software is not intended for safety control tasks! ***
 ***                       For further information see Comment tab!                        ***
 *********************************************************************************************)

IF sv_bInitStart THEN
   //register begin of inject sequence
   abBeginInjSequenceRegister.aRegister(@sv_MoveBeginInjectSequence);

   //register end of inject sequence
   abEndInjSequenceRegister.aRegister(@sv_MoveEndInjectSequence);

   //register begin of plast sequence
   abBeginPlastSequenceRegister.aRegister(@sv_MoveBeginPlastSequence);

   //register end of plast sequence
   abEndPlastSequenceRegister.aRegister(@sv_MoveEndPlastSequence);
END_IF;

;#END_EDIT_BLOCK END_ALGORITHM

POSTUPDATE_ALGORITHM pIntrusionMode ON PU_Task_7 WITH sv_IntrusionSettings.Mode

#BEGIN_EDIT_BLOCK
(**************************************** WARNING ********************************************
 *** The KEBA Kemro K2 System including software is not intended for safety control tasks! ***
 ***                       For further information see Comment tab!                        ***
 *********************************************************************************************)

//new sequence must be created
sv_bProgramSwitchChanged := TRUE;

;#END_EDIT_BLOCK END_ALGORITHM

POSTUPDATE_ALGORITHM pColdDrop ON PU_Task_7 WITH sv_ColdDropSettings.bUse

#BEGIN_EDIT_BLOCK
(**************************************** WARNING ********************************************
 *** The KEBA Kemro K2 System including software is not intended for safety control tasks! ***
 ***                       For further information see Comment tab!                        ***
 *********************************************************************************************)

//new sequence must be created
sv_bProgramSwitchChanged := TRUE;

;#END_EDIT_BLOCK END_ALGORITHM

POSTUPDATE_ALGORITHM pDurationChanged ON PU_Task_13 WITH sv_ColdDropSettings.dColdDropTime,sv_dDurationInjectAndHold

VAR
 fbUpdateProperties : FBUpdateEditorProperties;
END_VAR
#BEGIN_EDIT_BLOCK
(**************************************** WARNING ********************************************
 *** The KEBA Kemro K2 System including software is not intended for safety control tasks! ***
 ***                       For further information see Comment tab!                        ***
 *********************************************************************************************)

fbUpdateProperties();

;#END_EDIT_BLOCK END_ALGORITHM

POSTUPDATE_ALGORITHM pInjectActive ON PU_Task_13 WITH sv_bInjectActive

#BEGIN_EDIT_BLOCK
(**************************************** WARNING ********************************************
 *** The KEBA Kemro K2 System including software is not intended for safety control tasks! ***
 ***                       For further information see Comment tab!                        ***
 *********************************************************************************************)

IF NOT sv_bInjectActive THEN
   START_PROCESS_ALGORITHM(paResetHoldActive);
END_IF;

;#END_EDIT_BLOCK END_ALGORITHM

PROCESS_ALGORITHM paResetHoldActive ON TaskSlow

#BEGIN_EDIT_BLOCK
(**************************************** WARNING ********************************************
 *** The KEBA Kemro K2 System including software is not intended for safety control tasks! ***
 ***                       For further information see Comment tab!                        ***
 *********************************************************************************************)

//reset sv_bHoldActive after end of inject movement
//sv_bHoldActive is used as start condition reached flag if a parallel programmed
//movement refers to a detected CutOff instead of a position
//the slow task for resetting sv_bHoldActive is choosen to guarantee that also in
//the case of holding time is 0.0s a start condition reached information can be detected
//by the interpreter

sv_bHoldActive := FALSE;
STOP_PROCESS_ALGORITHM();

;#END_EDIT_BLOCK END_ALGORITHM

POSTUPDATE_ALGORITHM pDecompInstanceData ON PU_Task_7 WITH sv_InstanceDataDecompInterPos,sv_bInitDone

VAR_TEMP
 i : DINT;
END_VAR

VAR
 bInitDone : BOOL;
 PrevInstanceData : tyInstanceListArrayDecomp;
 bUpdate : BOOL;
 fbUpdateProperties : FBUpdateEditorProperties;
END_VAR
#BEGIN_EDIT_BLOCK
(**************************************** WARNING ********************************************
 *** The KEBA Kemro K2 System including software is not intended for safety control tasks! ***
 ***                       For further information see Comment tab!                        ***
 *********************************************************************************************)

IF NOT bInitDone THEN
   //save instance data after startup
   PrevInstanceData := sv_InstanceDataDecompInterPos;
   bInitDone := TRUE;
   RETURN;
END_IF;

FOR i := 1 TO cMaxIntermediateConditions DO

   bUpdate := FALSE;

   //copy set time to calculated duration
   //for representation in machine sequencer
   IF (sv_InstanceDataDecompInterPos[i].Mode = nDecompTimeDependent) AND
     (sv_InstanceDataDecompInterPos[i].dTime <> PrevInstanceData[i].dTime) THEN

      sv_InstanceDataDecompInterPos[i].dCalculatedDuration := sv_InstanceDataDecompInterPos[i].dTime;
      bUpdate := TRUE;
   END_IF;
END_FOR;

IF bUpdate THEN
   //trigger update of machine sequencer
   fbUpdateProperties();
END_IF;

;#END_EDIT_BLOCK END_ALGORITHM

POSTUPDATE_ALGORITHM pIntrusionProgrammed ON PU_Task_7 WITH sv_MoveIntrusion.bProgrammedInSequence

#BEGIN_EDIT_BLOCK
(**************************************** WARNING ********************************************
 *** The KEBA Kemro K2 System including software is not intended for safety control tasks! ***
 ***                       For further information see Comment tab!                        ***
 *********************************************************************************************)

IF NOT sv_bUseProgramSwitches THEN
   //sequence is programmed by editor
   //-> activate intrusion depending on the "programmed in sequence" information
   IF sv_MoveIntrusion.bProgrammedInSequence THEN
      sv_IntrusionSettings.Mode := nTimeDep;
   ELSE
      sv_IntrusionSettings.Mode := nNotUse;
   END_IF;
END_IF;

;#END_EDIT_BLOCK END_ALGORITHM

POSTUPDATE_ALGORITHM pColdDropProgrammed ON PU_Task_7 WITH sv_MoveColdDrop.bProgrammedInSequence

#BEGIN_EDIT_BLOCK
(**************************************** WARNING ********************************************
 *** The KEBA Kemro K2 System including software is not intended for safety control tasks! ***
 ***                       For further information see Comment tab!                        ***
 *********************************************************************************************)

IF NOT sv_bUseProgramSwitches THEN
   //sequence is programmed by editor
   //-> activate cold drop depending on the "programmed in sequence" information
   IF sv_MoveColdDrop.bProgrammedInSequence THEN
      sv_ColdDropSettings.bUse := TRUE;
   ELSE
      sv_ColdDropSettings.bUse := FALSE;
   END_IF;
END_IF;

;#END_EDIT_BLOCK END_ALGORITHM

END_ALGORITHM_BLOCK

#END_OF_IEC_PART

@Puma @IecEditor 6 97 @Pou 25
@@@BEG_Comment@@@
@h    ! WARNING !
@h    The Kemro K2 system (including software) only meets category B according to EN 954-1,
@h    thus it is not intended for usage in safety-relevant control applications in the field
@h    of personal safety (e.g. emergency stop).
@h    To implement potentially necessary safety-relevant control tasks, always use additional
@h    external safety devices that are intended for the particular purpose, and meet the necessary
@h    functional safety.
@h    For further information see EN 954-1 (EN ISO 13849-1) and/or the K2-x00 user manual, chapter
@h    "CE conformity, directives and standards".

Following functions are implemented in this AB
- registration of dummy movments for begin/end inject/plast sequence
- trigger new creation of machine sequence
- set/reset activated flags for intrusion and cold drop

@FunctionID: S_FU_05
@FunctionID: S_FU_04
@FunctionID: S_ALLG_09
@@@END_Comment@@@

@BEG_Contents

@BEG_Func
@RT(17)FuncTreeContainer
0
@END_Func

@BEG_Const
@RT(18)ConstTreeContainer
1
@Var @RT(26)cMaxIntermediateConditions @RT(0) @T @F @DT @RT(4)DINT @RT(0) @T @T @BASIC 0 @F
@F @F
@T
@BEG_Attrib
0 @RT(2)10 @RT(38)max. number of intermediate conditions
@END_Attrib
1 1 @F @F @F @F

@END_Const

@BEG_Export

@BEG_Kind
@ALGORITHM_BLOCK @RT(14)ABODCFunctions @STRUCTURED_TEXT
@RT(0) @RT(0) @RT(0)
@END_Kind

@BEG_Dcl
@RT(16)DclTreeContainer
19
@Var @RT(9)PU_Task_7 @RT(0) @T @F @DT @RT(4)TASK @RT(0) @T @T @BASIC 0 @F
@F @F
@T
@BEG_Attrib
3 @RT(0) @RT(0) @RT(0)
@END_Attrib
1 7 @F @F @F @F

@Var @RT(10)PU_Task_13 @RT(0) @T @F @DT @RT(4)TASK @RT(0) @T @T @BASIC 0 @F
@F @F
@T
@BEG_Attrib
3 @RT(0) @RT(0) @RT(0)
@END_Attrib
1 7 @F @F @F @F

@Var @RT(8)TaskSlow @RT(0) @T @F @DT @RT(4)TASK @RT(0) @T @T @BASIC 0 @F
@F @F
@T
@BEG_Attrib
3 @RT(0) @RT(0) @RT(0)
@END_Attrib
1 7 @F @F @F @F

@Var @RT(13)sv_bInitStart @RT(0) @T @F @DT @RT(4)BOOL @RT(0) @T @T @BASIC 0 @F
@F @F
@T
@BEG_Attrib
3 @RT(0) @RT(0) @RT(0)
@END_Attrib
1 8 @F @F @F @F

@Var @RT(26)sv_MoveBeginInjectSequence @RT(0) @T @T @DERIVED 0 @T @T @DT @RT(10)tsMoveData @RT(0) @T @T @UNKNOWN 0 @F
@F @F
@T
@BEG_Attrib
3 @RT(0) @RT(0) @RT(0)
@END_Attrib
1 8 @F @F @F @F

@Var @RT(24)sv_MoveEndInjectSequence @RT(0) @T @T @DERIVED 0 @T @T @DT @RT(10)tsMoveData @RT(0) @T @T @UNKNOWN 0 @F
@F @F
@T
@BEG_Attrib
3 @RT(0) @RT(0) @RT(0)
@END_Attrib
1 8 @F @F @F @F

@Var @RT(25)sv_MoveBeginPlastSequence @RT(0) @T @T @DERIVED 0 @T @T @DT @RT(10)tsMoveData @RT(0) @T @T @UNKNOWN 0 @F
@F @F
@T
@BEG_Attrib
3 @RT(0) @RT(0) @RT(0)
@END_Attrib
1 8 @F @F @F @F

@Var @RT(23)sv_MoveEndPlastSequence @RT(0) @T @T @DERIVED 0 @T @T @DT @RT(10)tsMoveData @RT(0) @T @T @UNKNOWN 0 @F
@F @F
@T
@BEG_Attrib
3 @RT(0) @RT(0) @RT(0)
@END_Attrib
1 8 @F @F @F @F

@Var @RT(20)sv_IntrusionSettings @RT(0) @T @T @DERIVED 0 @F @RT(16)tsIntrusionParam @F
@T
@BEG_Attrib
3 @RT(0) @RT(0) @RT(0)
@END_Attrib
1 8 @F @F @F @F

@Var @RT(24)sv_bProgramSwitchChanged @RT(0) @T @F @DT @RT(4)BOOL @RT(0) @T @T @BASIC 0 @F
@F @F
@T
@BEG_Attrib
3 @RT(0) @RT(77)TRUE if ODC sequence should be reinitialized because a program switch changed @RT(0)
@END_Attrib
1 8 @F @F @F @F

@Var @RT(19)sv_ColdDropSettings @RT(0) @T @T @DERIVED 0 @F @RT(16)tsColdDropParams @F
@T
@BEG_Attrib
3 @RT(0) @RT(0) @RT(0)
@END_Attrib
1 8 @F @F @F @F

@Var @RT(25)sv_dDurationInjectAndHold @RT(0) @T @F @DT @RT(4)TIME @RT(0) @T @T @BASIC 0 @F
@F @F
@T
@BEG_Attrib
3 @RT(0) @RT(25)Duration of inject + hold @RT(0)
@END_Attrib
1 8 @F @F @F @F

@Var @RT(14)sv_bHoldActive @RT(0) @T @F @DT @RT(4)BOOL @RT(0) @T @T @BASIC 0 @F
@F @F
@T
@BEG_Attrib
3 @RT(0) @RT(79)TRUE: holding is active; attention: SV is resetted after end of inject movement @RT(0)
@END_Attrib
1 8 @F @F @F @F

@Var @RT(16)sv_bInjectActive @RT(0) @T @F @DT @RT(4)BOOL @RT(0) @T @T @BASIC 0 @F
@F @F
@T
@BEG_Attrib
3 @RT(0) @RT(19)Injection is active @RT(0)
@END_Attrib
1 8 @F @F @F @F

@Var @RT(29)sv_InstanceDataDecompInterPos @RT(0) @T @T @DERIVED 0 @T @T @DT @RT(25)tyInstanceListArrayDecomp @RT(0) @T @T @UNKNOWN 0 @F
@F @F
@T
@BEG_Attrib
3 @RT(0) @RT(0) @RT(0)
@END_Attrib
1 8 @F @F @F @F

@Var @RT(12)sv_bInitDone @RT(0) @T @T @RENAMED 0 @T @T @DT @RT(4)BOOL @RT(0) @T @T @BASIC 0 @F
@F @F
@T
@BEG_Attrib
3 @RT(0) @RT(0) @RT(0)
@END_Attrib
1 8 @F @F @F @F

@Var @RT(16)sv_MoveIntrusion @RT(0) @T @T @DERIVED 0 @F @RT(10)tsMoveData @F
@T
@BEG_Attrib
3 @RT(0) @RT(0) @RT(0)
@END_Attrib
1 8 @F @F @F @F

@Var @RT(22)sv_bUseProgramSwitches @RT(0) @T @F @DT @RT(4)BOOL @RT(0) @T @T @BASIC 0 @F
@F @F
@T
@BEG_Attrib
3 @RT(0) @RT(84)TRUE: create sequence by using program switches; FALSE: use sequence from ODC editor @RT(0)
@END_Attrib
1 8 @F @F @F @F

@Var @RT(15)sv_MoveColdDrop @RT(0) @T @T @RENAMED 0 @T @T @DT @RT(10)tsMoveData @RT(0) @T @T @UNKNOWN 0 @F
@F @F
@T
@BEG_Attrib
3 @RT(0) @RT(0) @RT(0)
@END_Attrib
1 8 @F @F @F @F

@END_Dcl

@END_Export

@BEG_Body

9

@BEG_Export

@BEG_Algo
@POSTUPDATE_ALGORITHM @RT(10)pInitStart @STRUCTURED_TEXT
@RT(0) @RT(13)sv_bInitStart @RT(9)PU_Task_7 @F @F
@END_Algo

@BEG_Dcl
@RT(16)DclTreeContainer
4
@Var @RT(26)abBeginInjSequenceRegister @RT(0) @T @T @DERIVED 0 @T @T @DT @RT(18)ABMovementRegister @RT(0) @T @T @UNKNOWN 0 @F
@F @F
@T
@BEG_Attrib
3 @RT(0) @RT(0) @RT(0)
@END_Attrib
1 0 @F @F @F @F

@Var @RT(24)abEndInjSequenceRegister @RT(0) @T @T @DERIVED 0 @T @T @DT @RT(18)ABMovementRegister @RT(0) @T @T @UNKNOWN 0 @F
@F @F
@T
@BEG_Attrib
3 @RT(0) @RT(0) @RT(0)
@END_Attrib
1 0 @F @F @F @F

@Var @RT(28)abBeginPlastSequenceRegister @RT(0) @T @T @DERIVED 0 @T @T @DT @RT(18)ABMovementRegister @RT(0) @T @T @UNKNOWN 0 @F
@F @F
@T
@BEG_Attrib
3 @RT(0) @RT(0) @RT(0)
@END_Attrib
1 0 @F @F @F @F

@Var @RT(26)abEndPlastSequenceRegister @RT(0) @T @T @DERIVED 0 @T @T @DT @RT(18)ABMovementRegister @RT(0) @T @T @UNKNOWN 0 @F
@F @F
@T
@BEG_Attrib
3 @RT(0) @RT(0) @RT(0)
@END_Attrib
1 0 @F @F @F @F

@END_Dcl

@END_Export

@BEG_Export

@BEG_Algo
@POSTUPDATE_ALGORITHM @RT(14)pIntrusionMode @STRUCTURED_TEXT
@RT(0) @RT(25)sv_IntrusionSettings.Mode @RT(9)PU_Task_7 @F @F
@END_Algo

@BEG_Dcl
@RT(16)DclTreeContainer
0
@END_Dcl

@END_Export

@BEG_Export

@BEG_Algo
@POSTUPDATE_ALGORITHM @RT(9)pColdDrop @STRUCTURED_TEXT
@RT(0) @RT(24)sv_ColdDropSettings.bUse @RT(9)PU_Task_7 @F @F
@END_Algo

@BEG_Dcl
@RT(16)DclTreeContainer
0
@END_Dcl

@END_Export

@BEG_Export

@BEG_Algo
@POSTUPDATE_ALGORITHM @RT(16)pDurationChanged @STRUCTURED_TEXT
@RT(0) @RT(59)sv_ColdDropSettings.dColdDropTime,sv_dDurationInjectAndHold @RT(10)PU_Task_13 @F @F
@END_Algo

@BEG_Dcl
@RT(16)DclTreeContainer
1
@Var @RT(18)fbUpdateProperties @RT(0) @T @T @DERIVED 0 @T @T @DT @RT(24)FBUpdateEditorProperties @RT(0) @T @T @UNKNOWN 0 @F
@F @F
@T
@BEG_Attrib
3 @RT(0) @RT(0) @RT(0)
@END_Attrib
1 0 @F @F @F @F

@END_Dcl

@END_Export

@BEG_Export

@BEG_Algo
@POSTUPDATE_ALGORITHM @RT(13)pInjectActive @STRUCTURED_TEXT
@RT(0) @RT(16)sv_bInjectActive @RT(10)PU_Task_13 @F @F
@END_Algo

@BEG_Dcl
@RT(16)DclTreeContainer
0
@END_Dcl

@END_Export

@BEG_Export

@BEG_Algo
@PROCESS_ALGORITHM @RT(17)paResetHoldActive @STRUCTURED_TEXT
@RT(0) @RT(0) @RT(8)TaskSlow @F @F
@END_Algo

@BEG_Dcl
@RT(16)DclTreeContainer
0
@END_Dcl

@END_Export

@BEG_Export

@BEG_Algo
@POSTUPDATE_ALGORITHM @RT(19)pDecompInstanceData @STRUCTURED_TEXT
@RT(0) @RT(42)sv_InstanceDataDecompInterPos,sv_bInitDone @RT(9)PU_Task_7 @F @F
@END_Algo

@BEG_Dcl
@RT(16)DclTreeContainer
5
@Var @RT(9)bInitDone @RT(0) @T @F @DT @RT(4)BOOL @RT(0) @T @T @BASIC 0 @F
@F @F
@T
@BEG_Attrib
3 @RT(0) @RT(0) @RT(0)
@END_Attrib
1 0 @F @F @F @F

@Var @RT(16)PrevInstanceData @RT(0) @T @T @DERIVED 0 @T @T @DT @RT(25)tyInstanceListArrayDecomp @RT(0) @T @T @UNKNOWN 0 @F
@F @F
@T
@BEG_Attrib
3 @RT(0) @RT(0) @RT(0)
@END_Attrib
1 0 @F @F @F @F

@Var @RT(1)i @RT(0) @T @T @RENAMED 0 @T @T @DT @RT(4)DINT @RT(0) @T @T @BASIC 0 @F
@F @F
@T
@BEG_Attrib
3 @RT(0) @RT(0) @RT(0)
@END_Attrib
1 4 @F @F @F @F

@Var @RT(7)bUpdate @RT(0) @T @F @DT @RT(4)BOOL @RT(0) @T @T @BASIC 0 @F
@F @F
@T
@BEG_Attrib
3 @RT(0) @RT(0) @RT(0)
@END_Attrib
1 0 @F @F @F @F

@Var @RT(18)fbUpdateProperties @RT(0) @T @T @DERIVED 0 @T @T @DT @RT(24)FBUpdateEditorProperties @RT(0) @T @T @UNKNOWN 0 @F
@F @F
@T
@BEG_Attrib
3 @RT(0) @RT(0) @RT(0)
@END_Attrib
1 0 @F @F @F @F

@END_Dcl

@END_Export

@BEG_Export

@BEG_Algo
@POSTUPDATE_ALGORITHM @RT(20)pIntrusionProgrammed @STRUCTURED_TEXT
@RT(0) @RT(38)sv_MoveIntrusion.bProgrammedInSequence @RT(9)PU_Task_7 @F @F
@END_Algo

@BEG_Dcl
@RT(16)DclTreeContainer
0
@END_Dcl

@END_Export

@BEG_Export

@BEG_Algo
@POSTUPDATE_ALGORITHM @RT(19)pColdDropProgrammed @STRUCTURED_TEXT
@RT(0) @RT(37)sv_MoveColdDrop.bProgrammedInSequence @RT(9)PU_Task_7 @F @F
@END_Algo

@BEG_Dcl
@RT(16)DclTreeContainer
0
@END_Dcl

@END_Export

@BEG_Body
@TL(19)
(**************************************** WARNING ********************************************
 *** The KEBA Kemro K2 System including software is not intended for safety control tasks! ***
 ***                       For further information see Comment tab!                        ***
 *********************************************************************************************)

IF sv_bInitStart THEN
   //register begin of inject sequence
   abBeginInjSequenceRegister.aRegister(@sv_MoveBeginInjectSequence);

   //register end of inject sequence
   abEndInjSequenceRegister.aRegister(@sv_MoveEndInjectSequence);

   //register begin of plast sequence
   abBeginPlastSequenceRegister.aRegister(@sv_MoveBeginPlastSequence);

   //register end of plast sequence
   abEndPlastSequenceRegister.aRegister(@sv_MoveEndPlastSequence);
END_IF;

@END_Body

@@@BEG_Comment@@@
@TL(5)
registers the following dummy - movements:
- begin of inject sequence
- end of inject sequence
- begin of plast sequence
- end of plast sequence
@@@END_Comment@@@

@BEG_Body
@TL(8)
(**************************************** WARNING ********************************************
 *** The KEBA Kemro K2 System including software is not intended for safety control tasks! ***
 ***                       For further information see Comment tab!                        ***
 *********************************************************************************************)

//new sequence must be created
sv_bProgramSwitchChanged := TRUE;

@END_Body

@@@BEG_Comment@@@
@TL(0)

@@@END_Comment@@@

@BEG_Body
@TL(8)
(**************************************** WARNING ********************************************
 *** The KEBA Kemro K2 System including software is not intended for safety control tasks! ***
 ***                       For further information see Comment tab!                        ***
 *********************************************************************************************)

//new sequence must be created
sv_bProgramSwitchChanged := TRUE;

@END_Body

@@@BEG_Comment@@@
@TL(0)

@@@END_Comment@@@

@BEG_Body
@TL(7)
(**************************************** WARNING ********************************************
 *** The KEBA Kemro K2 System including software is not intended for safety control tasks! ***
 ***                       For further information see Comment tab!                        ***
 *********************************************************************************************)

fbUpdateProperties();

@END_Body

@@@BEG_Comment@@@
@TL(0)

@@@END_Comment@@@

@BEG_Body
@TL(11)
(**************************************** WARNING ********************************************
 *** The KEBA Kemro K2 System including software is not intended for safety control tasks! ***
 ***                       For further information see Comment tab!                        ***
 *********************************************************************************************)

IF NOT sv_bInjectActive THEN
   START_PROCESS_ALGORITHM(paResetHoldActive);
END_IF;

@END_Body

@@@BEG_Comment@@@
@TL(0)

@@@END_Comment@@@

@BEG_Body
@TL(15)
(**************************************** WARNING ********************************************
 *** The KEBA Kemro K2 System including software is not intended for safety control tasks! ***
 ***                       For further information see Comment tab!                        ***
 *********************************************************************************************)

//reset sv_bHoldActive after end of inject movement
//sv_bHoldActive is used as start condition reached flag if a parallel programmed
//movement refers to a detected CutOff instead of a position
//the slow task for resetting sv_bHoldActive is choosen to guarantee that also in
//the case of holding time is 0.0s a start condition reached information can be detected
//by the interpreter

sv_bHoldActive := FALSE;
STOP_PROCESS_ALGORITHM();

@END_Body

@@@BEG_Comment@@@
@TL(0)

@@@END_Comment@@@

@BEG_Body
@TL(32)
(**************************************** WARNING ********************************************
 *** The KEBA Kemro K2 System including software is not intended for safety control tasks! ***
 ***                       For further information see Comment tab!                        ***
 *********************************************************************************************)

IF NOT bInitDone THEN
   //save instance data after startup
   PrevInstanceData := sv_InstanceDataDecompInterPos;
   bInitDone := TRUE;
   RETURN;
END_IF;

FOR i := 1 TO cMaxIntermediateConditions DO

   bUpdate := FALSE;

   //copy set time to calculated duration
   //for representation in machine sequencer
   IF (sv_InstanceDataDecompInterPos[i].Mode = nDecompTimeDependent) AND
     (sv_InstanceDataDecompInterPos[i].dTime <> PrevInstanceData[i].dTime) THEN

      sv_InstanceDataDecompInterPos[i].dCalculatedDuration := sv_InstanceDataDecompInterPos[i].dTime;
      bUpdate := TRUE;
   END_IF;
END_FOR;

IF bUpdate THEN
   //trigger update of machine sequencer
   fbUpdateProperties();
END_IF;

@END_Body

@@@BEG_Comment@@@
@TL(0)

@@@END_Comment@@@

@BEG_Body
@TL(15)
(**************************************** WARNING ********************************************
 *** The KEBA Kemro K2 System including software is not intended for safety control tasks! ***
 ***                       For further information see Comment tab!                        ***
 *********************************************************************************************)

IF NOT sv_bUseProgramSwitches THEN
   //sequence is programmed by editor
   //-> activate intrusion depending on the "programmed in sequence" information
   IF sv_MoveIntrusion.bProgrammedInSequence THEN
      sv_IntrusionSettings.Mode := nTimeDep;
   ELSE
      sv_IntrusionSettings.Mode := nNotUse;
   END_IF;
END_IF;

@END_Body

@@@BEG_Comment@@@
@TL(0)

@@@END_Comment@@@

@BEG_Body
@TL(15)
(**************************************** WARNING ********************************************
 *** The KEBA Kemro K2 System including software is not intended for safety control tasks! ***
 ***                       For further information see Comment tab!                        ***
 *********************************************************************************************)

IF NOT sv_bUseProgramSwitches THEN
   //sequence is programmed by editor
   //-> activate cold drop depending on the "programmed in sequence" information
   IF sv_MoveColdDrop.bProgrammedInSequence THEN
      sv_ColdDropSettings.bUse := TRUE;
   ELSE
      sv_ColdDropSettings.bUse := FALSE;
   END_IF;
END_IF;

@END_Body

@@@BEG_Comment@@@
@TL(0)

@@@END_Comment@@@
@END_Body

@END_Contents

(* ---- ABOutElectricPlast.pu ---- *)
(*
@h    ! WARNING !
@h    The Kemro K2 system (including software) only meets category B according to EN 954-1,
@h    thus it is not intended for usage in safety-relevant control applications in the field
@h    of personal safety (e.g. emergency stop).
@h    To implement potentially necessary safety-relevant control tasks, always use additional
@h    external safety devices that are intended for the particular purpose, and meet the necessary
@h    functional safety.
@h    For further information see EN 954-1 (EN ISO 13849-1) and/or the K2-x00 user manual, chapter
@h    "CE conformity, directives and standards".

analog output to electric plast motor

@FunctionID: CR_0033583

*)

IMPORT_OVER_LISTFILE
 nElectric
, nHydraulic
, cMovePlast
, cMoveIntrusion
, cMovePlastPurge
, tnMotorType
, tsMoveCtrl
, ABAnalogHWOut
, tnDataState

END_IMPORT

ALGORITHM_BLOCK ABOutElectricPlast #DUMMY_EDIT_BLOCK

SYSTEM_VAR
 sv_bPreOutputReady : BOOL (* PreOutput is ready *);
 sv_bInitStart : BOOL (* Device registration finished - custom IEC initialisation can be started *);
 sv_PlastMotor : tnMotorType (* type of plast motor *);
 sv_bOutputActive : BOOL (* Output is active *);
 sv_rVelocity : REAL (* set value for velocity *);
 sv_DataState : tnDataState;
END_VAR

SYSTEM_OBJECT
 PU_Task_7 : TASK;
 TaskAnalog : TASK;
END_OBJECT

VAR_EXTERNAL
 g_MoveCtrl : tsMoveCtrl;
END_VAR

VAR
 abAnalogOut : ABAnalogHWOut;
END_VAR

POSTUPDATE_ALGORITHM pDataState ON PU_Task_7 WITH sv_DataState

VAR
 bMDLoadingInProgress : BOOL (* loading of machine data in progress *);
END_VAR
#BEGIN_EDIT_BLOCK
(**************************************** WARNING ********************************************
 *** The KEBA Kemro K2 System including software is not intended for safety control tasks! ***
 ***                       For further information see Comment tab!                        ***
 *********************************************************************************************)

IF sv_DataState = nReadMachineData THEN
   //loading of machinedata in progress
   bMDLoadingInProgress := TRUE;
   RETURN;
END_IF;

IF sv_DataState = nReady AND bMDLoadingInProgress THEN

   //set sv_PlastMotor after loading of machine data
   IF (abAnalogOut.aIsLinked()) THEN
      sv_PlastMotor := nElectric;
   ELSE
      sv_PlastMotor := nHydraulic;
   END_IF;

   bMDLoadingInProgress := FALSE;
END_IF;

;#END_EDIT_BLOCK END_ALGORITHM

POSTUPDATE_ALGORITHM pCheckMode ON PU_Task_7 WITH sv_bInitStart

#BEGIN_EDIT_BLOCK
(**************************************** WARNING ********************************************
 *** The KEBA Kemro K2 System including software is not intended for safety control tasks! ***
 ***                       For further information see Comment tab!                        ***
 *********************************************************************************************)

IF (abAnalogOut.aIsLinked()) THEN
    sv_PlastMotor := nElectric;
ELSE
    sv_PlastMotor := nHydraulic;
END_IF;

;#END_EDIT_BLOCK END_ALGORITHM

PROCESS_ALGORITHM paRun ON TaskAnalog

(* IecGraph-Code *)

(* init step *)
INITIAL_STEP START:
END_STEP

(* steps *)
STEP Step20:
Action21 (N);
END_STEP

ACTION Action21: #BEGIN_EDIT_BLOCK
abAnalogOut.aOut(sv_rVelocity/10.0);

;#END_EDIT_BLOCK END_ACTION (*Action21*)
STEP END:
Action3 (P);
END_STEP

ACTION Action3: #BEGIN_EDIT_BLOCK
abAnalogOut.aOut(0.0);
STOP_PROCESS_ALGORITHM();

;#END_EDIT_BLOCK END_ACTION (*Action3*)

(* transitions *)
GO_ON_TRANSITION Trans32 (* Trans32 *) FROM START TO Step20 :=  #BEGIN_EDIT_BLOCK
sv_bPreOutputReady AND
sv_bOutputActive
;#END_EDIT_BLOCK
END_TRANSITION

GO_ON_TRANSITION Trans33 (* Trans33 *) FROM START TO END :=  #BEGIN_EDIT_BLOCK
NOT sv_bOutputActive
;#END_EDIT_BLOCK
END_TRANSITION

GO_ON_TRANSITION Trans34 (* Trans34 *) FROM Step20 TO END :=  #BEGIN_EDIT_BLOCK
NOT sv_bOutputActive
;#END_EDIT_BLOCK
END_TRANSITION

TRANSITION Trans16 (* Trans16 *) FROM END TO START :=  #BEGIN_EDIT_BLOCK
TRUE
;#END_EDIT_BLOCK
END_TRANSITION

(* end IecGraph-Code *)
(* sfc-code *)
(* end sfc-code *)

END_ALGORITHM

POSTUPDATE_ALGORITHM pOutputActive ON PU_Task_7 WITH sv_bOutputActive

#BEGIN_EDIT_BLOCK
IF sv_bOutputActive THEN
    IF  (((g_MoveCtrl.pData^.MoveId = cMovePlast)
            OR (g_MoveCtrl.pData^.MoveId = cMoveIntrusion)
            OR (g_MoveCtrl.pData^.MoveId = cMovePlastPurge))
        AND (sv_PlastMotor = nElectric)) THEN
        START_PROCESS_ALGORITHM(paRun);
    END_IF;
END_IF;

;#END_EDIT_BLOCK END_ALGORITHM

END_ALGORITHM_BLOCK

#END_OF_IEC_PART

@Puma @IecEditor 6 114 @Pou 25
@@@BEG_Comment@@@
@h    ! WARNING !
@h    The Kemro K2 system (including software) only meets category B according to EN 954-1,
@h    thus it is not intended for usage in safety-relevant control applications in the field
@h    of personal safety (e.g. emergency stop).
@h    To implement potentially necessary safety-relevant control tasks, always use additional
@h    external safety devices that are intended for the particular purpose, and meet the necessary
@h    functional safety.
@h    For further information see EN 954-1 (EN ISO 13849-1) and/or the K2-x00 user manual, chapter
@h    "CE conformity, directives and standards".

analog output to electric plast motor

@FunctionID: CR_0033583

@@@END_Comment@@@

@BEG_Contents

@BEG_Func
@RT(17)FuncTreeContainer
0
@END_Func

@BEG_Const
@RT(18)ConstTreeContainer
5
@Var @RT(9)nElectric @RT(0) @T @T @DERIVED 0 @F @RT(11)tnMotorType @F
@T
@BEG_Attrib
0 @RT(1)1 @RT(14)electric motor
@END_Attrib
1 1 @F @F @F @F

@Var @RT(10)nHydraulic @RT(0) @T @T @DERIVED 0 @F @RT(11)tnMotorType @F
@T
@BEG_Attrib
0 @RT(1)0 @RT(15)hydraulic motor
@END_Attrib
1 1 @F @F @F @F

@Var @RT(10)cMovePlast @RT(0) @T @F @DT @RT(4)DINT @RT(0) @T @T @BASIC 0 @F
@F @F
@T
@BEG_Attrib
0 @RT(2)13 @RT(23)plast movement (rotate)
@END_Attrib
1 1 @F @F @F @F

@Var @RT(14)cMoveIntrusion @RT(0) @T @F @DT @RT(4)DINT @RT(0) @T @T @BASIC 0 @F
@F @F
@T
@BEG_Attrib
0 @RT(2)28 @RT(9)intrusion
@END_Attrib
1 1 @F @F @F @F

@Var @RT(15)cMovePlastPurge @RT(0) @T @F @DT @RT(4)DINT @RT(0) @T @T @BASIC 0 @F
@F @F
@T
@BEG_Attrib
0 @RT(2)34 @RT(26)plast movement for purging
@END_Attrib
1 1 @F @F @F @F

@END_Const

@BEG_Export

@BEG_Kind
@ALGORITHM_BLOCK @RT(18)ABOutElectricPlast @STRUCTURED_TEXT
@RT(0) @RT(0) @RT(0)
@END_Kind

@BEG_Dcl
@RT(16)DclTreeContainer
10
@Var @RT(18)sv_bPreOutputReady @RT(0) @T @F @DT @RT(4)BOOL @RT(0) @T @T @BASIC 0 @F
@F @F
@T
@BEG_Attrib
3 @RT(0) @RT(18)PreOutput is ready @RT(0)
@END_Attrib
1 8 @F @F @F @F

@Var @RT(13)sv_bInitStart @RT(0) @T @F @DT @RT(4)BOOL @RT(0) @T @T @BASIC 0 @F
@F @F
@T
@BEG_Attrib
3 @RT(0) @RT(71)Device registration finished - custom IEC initialisation can be started @RT(0)
@END_Attrib
1 8 @F @F @F @F

@Var @RT(13)sv_PlastMotor @RT(0) @T @T @DERIVED 0 @T @T @DT @RT(11)tnMotorType @RT(0) @T @T @UNKNOWN 0 @F
@F @F
@T
@BEG_Attrib
3 @RT(0) @RT(19)type of plast motor @RT(0)
@END_Attrib
1 8 @F @F @F @F

@Var @RT(16)sv_bOutputActive @RT(0) @T @F @DT @RT(4)BOOL @RT(0) @T @T @BASIC 0 @F
@F @F
@T
@BEG_Attrib
3 @RT(0) @RT(16)Output is active @RT(0)
@END_Attrib
1 8 @F @F @F @F

@Var @RT(12)sv_rVelocity @RT(0) @T @F @DT @RT(4)REAL @RT(0) @T @T @BASIC 0 @F
@F @F
@T
@BEG_Attrib
3 @RT(0) @RT(22)set value for velocity @RT(0)
@END_Attrib
1 8 @F @F @F @F

@Var @RT(9)PU_Task_7 @RT(0) @T @F @DT @RT(4)TASK @RT(0) @T @T @BASIC 0 @F
@F @F
@T
@BEG_Attrib
3 @RT(0) @RT(0) @RT(0)
@END_Attrib
1 7 @F @F @F @F

@Var @RT(10)TaskAnalog @RT(0) @T @F @DT @RT(4)TASK @RT(0) @T @T @BASIC 0 @F
@F @F
@T
@BEG_Attrib
3 @RT(0) @RT(0) @RT(0)
@END_Attrib
1 7 @F @F @F @F

@Var @RT(10)g_MoveCtrl @RT(0) @T @T @DERIVED 0 @T @T @DT @RT(10)tsMoveCtrl @RT(0) @T @T @UNKNOWN 0 @F
@F @F
@T
@BEG_Attrib
3 @RT(0) @RT(0) @RT(0)
@END_Attrib
1 6 @F @F @F @F

@Var @RT(11)abAnalogOut @RT(0) @T @T @DERIVED 0 @T @T @DT @RT(13)ABAnalogHWOut @RT(0) @T @T @UNKNOWN 0 @F
@F @F
@T
@BEG_Attrib
3 @RT(0) @RT(0) @RT(0)
@END_Attrib
1 0 @F @F @F @F

@Var @RT(12)sv_DataState @RT(0) @T @T @DERIVED 0 @T @T @DT @RT(11)tnDataState @RT(0) @T @T @UNKNOWN 0 @F
@F @F
@T
@BEG_Attrib
3 @RT(0) @RT(0) @RT(0)
@END_Attrib
1 8 @F @F @F @F

@END_Dcl

@END_Export

@BEG_Body

4

@BEG_Export

@BEG_Algo
@POSTUPDATE_ALGORITHM @RT(10)pDataState @STRUCTURED_TEXT
@RT(0) @RT(12)sv_DataState @RT(9)PU_Task_7 @F @F
@END_Algo

@BEG_Dcl
@RT(16)DclTreeContainer
1
@Var @RT(20)bMDLoadingInProgress @RT(0) @T @F @DT @RT(4)BOOL @RT(0) @T @T @BASIC 0 @F
@F @F
@T
@BEG_Attrib
3 @RT(0) @RT(35)loading of machine data in progress @RT(0)
@END_Attrib
1 0 @F @F @F @F

@END_Dcl

@END_Export

@BEG_Export

@BEG_Algo
@POSTUPDATE_ALGORITHM @RT(10)pCheckMode @STRUCTURED_TEXT
@RT(0) @RT(13)sv_bInitStart @RT(9)PU_Task_7 @F @F
@END_Algo

@BEG_Dcl
@RT(16)DclTreeContainer
0
@END_Dcl

@END_Export

@BEG_Export

@BEG_Algo
@PROCESS_ALGORITHM @RT(5)paRun @SEQUENTIAL_FLOW_CHART
@RT(0) @RT(0) @RT(10)TaskAnalog @F @F
@END_Algo

@BEG_Dcl
@RT(16)DclTreeContainer
0
@END_Dcl

@END_Export

@BEG_Export

@BEG_Algo
@POSTUPDATE_ALGORITHM @RT(13)pOutputActive @STRUCTURED_TEXT
@RT(0) @RT(16)sv_bOutputActive @RT(9)PU_Task_7 @F @F
@END_Algo

@BEG_Dcl
@RT(16)DclTreeContainer
0
@END_Dcl

@END_Export

@BEG_Body
@TL(25)
(**************************************** WARNING ********************************************
 *** The KEBA Kemro K2 System including software is not intended for safety control tasks! ***
 ***                       For further information see Comment tab!                        ***
 *********************************************************************************************)

IF sv_DataState = nReadMachineData THEN
   //loading of machinedata in progress
   bMDLoadingInProgress := TRUE;
   RETURN;
END_IF;

IF sv_DataState = nReady AND bMDLoadingInProgress THEN

   //set sv_PlastMotor after loading of machine data
   IF (abAnalogOut.aIsLinked()) THEN
      sv_PlastMotor := nElectric;
   ELSE
      sv_PlastMotor := nHydraulic;
   END_IF;

   bMDLoadingInProgress := FALSE;
END_IF;

@END_Body

@@@BEG_Comment@@@
@TL(0)

@@@END_Comment@@@

@BEG_Body
@TL(11)
(**************************************** WARNING ********************************************
 *** The KEBA Kemro K2 System including software is not intended for safety control tasks! ***
 ***                       For further information see Comment tab!                        ***
 *********************************************************************************************)

IF (abAnalogOut.aIsLinked()) THEN
    sv_PlastMotor := nElectric;
ELSE
    sv_PlastMotor := nHydraulic;
END_IF;

@END_Body

@@@BEG_Comment@@@
@TL(0)

@@@END_Comment@@@

@BEG_SfcBody
3 5 5

@BEG_SfcData 2
@StepSeq @RT(4)sseq @F 1
@Loop @RT(4)loop @F 2
@StepSeq @RT(4)sseq @F 5
@Step @RT(5)START @F @T @F @F @RT(0) @F
@AcbCont @RT(7)unnamed @F 0

@AltBranch @RT(3)alt @F 2
@TransSeq @RT(4)tseq @F 1
@Trans @RT(7)Trans32 @F @T @F @F @T @F @TL(3)
sv_bPreOutputReady AND
sv_bOutputActive

@RT(7)Trans32 @F

@TransSeq @RT(4)tseq @F 2
@Trans @RT(7)Trans33 @F @T @F @F @T @F @TL(2)
NOT sv_bOutputActive

@RT(7)Trans33 @F
@Goto @RT(3)END @F @F

@Step @RT(6)Step20 @F @F @F @F @RT(0) @F
@AcbCont @RT(7)unnamed @F 1
@Acb @RT(8)Action21 @F @T @RT(1)N @RT(0) @F @F @T @TL(2)
abAnalogOut.aOut(sv_rVelocity/10.0);

@F

@Trans @RT(7)Trans34 @F @T @F @F @T @F @TL(2)
NOT sv_bOutputActive

@RT(7)Trans34 @F
@Step @RT(3)END @F @F @T @F @RT(0) @F
@AcbCont @RT(7)unnamed @F 1
@Acb @RT(7)Action3 @F @T @RT(1)P @RT(0) @F @F @T @TL(3)
abAnalogOut.aOut(0.0);
STOP_PROCESS_ALGORITHM();

@F

@Trans @RT(7)Trans16 @F @T @F @T @T @T @TL(2)
TRUE

@RT(7)Trans16 @F

@END_SfcData
@SaActions 0
@SaTrans 0
@SaExits 0
@END_SfcBody

@@@BEG_Comment@@@
@TL(0)

@@@END_Comment@@@

@BEG_Body
@TL(9)
IF sv_bOutputActive THEN
    IF  (((g_MoveCtrl.pData^.MoveId = cMovePlast)
            OR (g_MoveCtrl.pData^.MoveId = cMoveIntrusion)
            OR (g_MoveCtrl.pData^.MoveId = cMovePlastPurge))
        AND (sv_PlastMotor = nElectric)) THEN
        START_PROCESS_ALGORITHM(paRun);
    END_IF;
END_IF;

@END_Body

@@@BEG_Comment@@@
@TL(0)

@@@END_Comment@@@
@END_Body

@END_Contents
